FUNCTION ACFrequencyCheck : BOOL
VAR_INPUT
	IN			: REAL;
END_VAR
VAR
	r_min		: REAL;
	r_max		: REAL;
END_VAR

r_min:= settings.GridParams.r_GridFrequencyMin;
r_max:= settings.GridParams.r_GridFrequencyMax;

ACfrequencyCheck := LIMIT(r_min, IN, r_max) = IN;

END_FUNCTION

(* stored: Version 1.1.0.1, ProductVersion 3.1.4026.18
   POU ACFrequencyCheck: Id {e2a791e4-e151-4de0-9e10-9102876dee16}, SpecialFunc None *)
